{attribute 'qualified_only'}
{attribute 'strict'}
TYPE E_IODEV_ERROR :
(
	OK					:= 0,
	HW_NOT_OP			:= 1,			
	WRONG_CMD			:= 2,			
	INIT_FAILURE		:= 3,		

	NOT_INITIALISED		:= 90,
	ZERO_POINTER		:= 100	// Simulator error
);
END_TYPE

(* stored: Version 1.1.0.1, ProductVersion 3.1.4022.16
   DUT E_IODEV_ERROR: Id {4921bf0b-46a2-4adb-9997-96612de65a31} *)
